// Mitsubishi GX Works2 project: 0708_P_002_conAdded   PLC: Q03UDV

// global labels: Global1
VAR_GLOBAL
  R흡착기온명령 AT X1000 : BOOL;
  R흡착기오프명령 AT X1001 : BOOL;
  흡착기온솔밸브 AT Y42 : BOOL;
  흡착기오프솔밸브 AT Y43 : BOOL;
  TG1 AT X2A : BOOL;
  TG2 AT X2B : BOOL;
  TG3 AT X2C : BOOL;
  PB4 AT X2D : BOOL;
  PB5 AT X2E : BOOL;
  경광녹색 AT Y44 : BOOL;
  경광황색 AT Y45 : BOOL;
  경광적색 AT Y46 : BOOL;
  부저 AT Y47 : BOOL;
  컨베이어_정구동 AT Y48 : BOOL;
  컨베이어_역구동 AT Y49 : BOOL;
  R고정온명령 AT X1010 : BOOL;
  R고정오프명령 AT X1011 : BOOL;
  고정전솔 AT Y40 : BOOL;
  고정후솔 AT Y41 : BOOL;
END_VAR

PROGRAM MAIN
VAR
  컨베이어_정구동신호 : BOOL;
  컨베이어_역구동신호 : BOOL;
END_VAR
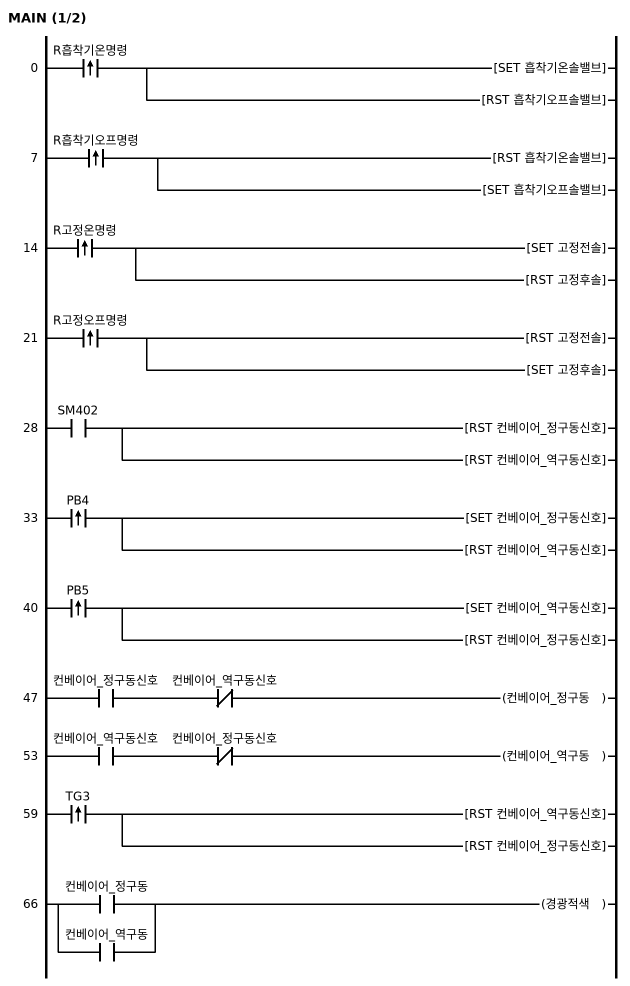
0     LDP     R흡착기온명령
      SET     흡착기온솔밸브
      RST     흡착기오프솔밸브
7     LDP     R흡착기오프명령
      RST     흡착기온솔밸브
      SET     흡착기오프솔밸브
14    LDP     R고정온명령
      SET     고정전솔
      RST     고정후솔
21    LDP     R고정오프명령
      RST     고정전솔
      SET     고정후솔
28    LD      SM402
      RST     컨베이어_정구동신호
      RST     컨베이어_역구동신호
33    LDP     PB4
      SET     컨베이어_정구동신호
      RST     컨베이어_역구동신호
40    LDP     PB5
      SET     컨베이어_역구동신호
      RST     컨베이어_정구동신호
47    LD      컨베이어_정구동신호
      ANI     컨베이어_역구동신호
      OUT     컨베이어_정구동
53    LD      컨베이어_역구동신호
      ANI     컨베이어_정구동신호
      OUT     컨베이어_역구동
59    LDP     TG3
      RST     컨베이어_역구동신호
      RST     컨베이어_정구동신호
66    LD      컨베이어_정구동
      OR      컨베이어_역구동
      OUT     경광적색
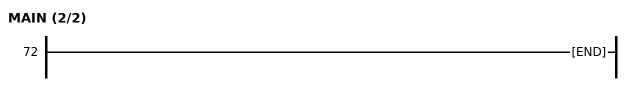
72    END
END_PROGRAM
